{attribute 'GeneratedUsingTerminal: AT2026-0250-0022'}
{attribute addProperty BoxType "AT2026-0250-0022"}
{attribute addProperty Id "A_0079_AT2002_5249_0018_AT2002_5249AT2002_01D6DEDF80"}
{attribute addProperty CRC "770534154"}
{attribute addProperty Size "80"}
TYPE A_0067_AT2026_0250_0022_AT2026_0250_2DED6B0A EXTENDS AT2026_86175B41 :
STRUCT
	{attribute addProperty Name "A_0079_AT2002_5249_0018_AT2002_5249"}
	{attribute addProperty PreviousPort "A_0067(AT2026-0250-0022) (AT2026-0250) : B"}
	A_0079_AT2002_5249_0018_AT2002_5249 : AT2002_01D6DEDF;
END_STRUCT
END_TYPE

(* stored: Version 1.2.0.0, ProductVersion 3.1.4024.9
   DUT A_0067_AT2026_0250_0022_AT2026_0250_2DED6B0A: Id {9d5fa4f2-53e0-4627-98ee-e1bb9c8a0bd4} *)
